                                               END_IF;
                                           END_FOR;
                                           //Beschränkung mögliche Nummer in dem Viereck 5
                                           #initial := 30;
                                           #länge := 32;
                                           FOR #m := 0 TO 2 BY 1 DO
                                               FOR #i := #initial TO #länge BY 1 DO
                                                   IF #gitter[#k].nummer > 0 THEN
                                                       #gitter[#i].potenz_nummer[#gitter[#k].nummer - 1] := FALSE;
                                                   END_IF;
                                               END_FOR;
                                               IF #m < 2 THEN
                                                   #initial := #initial + 9;
                                                   #länge := #länge + 9;
                                               END_IF;
                                           END_FOR;
                                       END_REGION
                                       //Feldchen 41
                                   40:
                                       REGION Feldchen 41
                                           //Beschränkung mögliche Nummer in der Zeile 5
                                           FOR #i := 36 TO 44 BY 1 DO
                                               IF #gitter[#k].nummer > 0 THEN
                                                   #gitter[#i].potenz_nummer[#gitter[#k].nummer - 1] := FALSE;
                                               END_IF;
                                           END_FOR;
                                           //Beschränkung mögliche Nummer in der Säule 5
                                           FOR #i := 4 TO 80 BY 9 DO
                                               IF #gitter[#k].nummer > 0 THEN
                                                   #gitter[#i].potenz_nummer[#gitter[#k].nummer - 1] := FALSE;
                                               END_IF;
                                           END_FOR;
                                           //Beschränkung mögliche Nummer in dem Viereck 5
                                           #initial := 30;
                                           #länge := 32;
                                           FOR #m := 0 TO 2 BY 1 DO
                                               FOR #i := #initial TO #länge BY 1 DO
                                                   IF #gitter[#k].nummer > 0 THEN
                                                       #gitter[#i].potenz_nummer[#gitter[#k].nummer - 1] := FALSE;
                                                   END_IF;
                                               END_FOR;
                                               IF #m < 2 THEN
                                                   #initial := #initial + 9;
                                                   #länge := #länge + 9;
                                               END_IF;
                                           END_FOR;
                                       END_REGION
                                       //Feldchen 42
                                   41:
                                       REGION Feldchen 42
                                           //Beschränkung mögliche Nummer in der Zeile 5
                                           FOR #i := 36 TO 44 BY 1 DO
                                               IF #gitter[#k].nummer > 0 THEN
                                                   #gitter[#i].potenz_nummer[#gitter[#k].nummer - 1] := FALSE;
                                               END_IF;
                                           END_FOR;
                                           //Beschränkung mögliche Nummer in der Säule 6
                                           FOR #i := 5 TO 80 BY 9 DO
                                               IF #gitter[#k].nummer > 0 THEN
                                                   #gitter[#i].potenz_nummer[#gitter[#k].nummer - 1] := FALSE;
                                               END_IF;
                                           END_FOR;
                                           //Beschränkung mögliche Nummer in dem Viereck 5
                                           #initial := 30;
                                           #länge := 32;
                                           FOR #m := 0 TO 2 BY 1 DO
                                               FOR #i := #initial TO #länge BY 1 DO
                                                   IF #gitter[#k].nummer > 0 THEN
                                                       #gitter[#i].potenz_nummer[#gitter[#k].nummer - 1] := FALSE;
                                                   END_IF;
                                               END_FOR;
                                               IF #m < 2 THEN
                                                   #initial := #initial + 9;
                                                   #länge := #länge + 9;
                                               END_IF;
                                           END_FOR;
                                       END_REGION
                                       //Feldchen 43
                                   42:
                                       REGION Feldchen 43
                                           //Beschränkung mögliche Nummer in der Zeile 5
                                           FOR #i := 36 TO 44 BY 1 DO
                                               IF #gitter[#k].nummer > 0 THEN
                                                   #gitter[#i].potenz_nummer[#gitter[#k].nummer - 1] := FALSE;
                                               END_IF;
                                           END_FOR;
                                           //Beschränkung mögliche Nummer in der Säule 7
                                           FOR #i := 6 TO 80 BY 9 DO
                                               IF #gitter[#k].nummer > 0 THEN
                                                   #gitter[#i].potenz_nummer[#gitter[#k].nummer - 1] := FALSE;
                                               END_IF;
                                           END_FOR;
                                           //Beschränkung mögliche Nummer in dem Viereck 6
                                           #initial := 33;
                                           #länge := 35;
                                           FOR #m := 0 TO 2 BY 1 DO
                                               FOR #i := #initial TO #länge BY 1 DO
                                                   IF #gitter[#k].nummer > 0 THEN
                                                       #gitter[#i].potenz_nummer[#gitter[#k].nummer - 1] := FALSE;
                                                   END_IF;
                                               END_FOR;
                                               IF #m < 2 THEN
                                                   #initial := #initial + 9;
                                                   #länge := #länge + 9;
                                               END_IF;
                                           END_FOR;
                                       END_REGION
                                       //Feldchen 44
                                   43:
                                       REGION Feldchen 44
                                           //Beschränkung mögliche Nummer in der Zeile 5
                                           FOR #i := 36 TO 44 BY 1 DO
                                               IF #gitter[#k].nummer > 0 THEN
                                                   #gitter[#i].potenz_nummer[#gitter[#k].nummer - 1] := FALSE;
                                               END_IF;
                                           END_FOR;
                                           //Beschränkung mögliche Nummer in der Säule 8
                                           FOR #i := 7 TO 80 BY 9 DO
                                               IF #gitter[#k].nummer > 0 THEN
                                                   #gitter[#i].potenz_nummer[#gitter[#k].nummer - 1] := FALSE;
                                               END_IF;
                                           END_FOR;
                                           //Beschränkung mögliche Nummer in dem Viereck 6
                                           #initial := 33;
                                           #länge := 35;
                                           FOR #m := 0 TO 2 BY 1 DO
                                               FOR #i := #initial TO #länge BY 1 DO
                                                   IF #gitter[#k].nummer > 0 THEN
                                                       #gitter[#i].potenz_nummer[#gitter[#k].nummer - 1] := FALSE;
                                                   END_IF;
                                               END_FOR;
                                               IF #m < 2 THEN
                                                   #initial := #initial + 9;
                                                   #länge := #länge + 9;
                                               END_IF;
                                           END_FOR;
                                       END_REGION
                                       //Feldchen 45
                                   44:
                                       REGION Feldchen 45
                                           //Beschränkung mögliche Nummer in der Zeile 5
                                           FOR #i := 36 TO 44 BY 1 DO
                                               IF #gitter[#k].nummer > 0 THEN
                                                   #gitter[#i].potenz_nummer[#gitter[#k].nummer - 1] := FALSE;
                                               END_IF;
                                           END_FOR;
                                           //Beschränkung mögliche Nummer in der Säule 9
                                           FOR #i := 8 TO 80 BY 9 DO
                                               IF #gitter[#k].nummer > 0 THEN
                                                   #gitter[#i].potenz_nummer[#gitter[#k].nummer - 1] := FALSE;
                                               END_IF;
                                           END_FOR;
                                           //Beschränkung mögliche Nummer in dem Viereck 6
                                           #initial := 33;
                                           #länge := 35;
                                           FOR #m := 0 TO 2 BY 1 DO
                                               FOR #i := #initial TO #länge BY 1 DO
                                                   IF #gitter[#k].nummer > 0 THEN
                                                       #gitter[#i].potenz_nummer[#gitter[#k].nummer - 1] := FALSE;
                                                   END_IF;
                                               END_FOR;
                                               IF #m < 2 THEN
                                                   #initial := #initial + 9;
                                                   #länge := #länge + 9;
                                               END_IF;
                                           END_FOR;
                                       END_REGION
                                       //Feldchen 46
                                   45:
                                       REGION Feldchen 46
                                           //Beschränkung mögliche Nummer in der Zeile 6
                                           FOR #i := 45 TO 53 BY 1 DO
                                               IF #gitter[#k].nummer > 0 THEN
                                                   #gitter[#i].potenz_nummer[#gitter[#k].nummer - 1] := FALSE;
                                               END_IF;
                                           END_FOR;
                                           //Beschränkung mögliche Nummer in der Säule 1
                                           FOR #i := 0 TO 80 BY 9 DO
                                               IF #gitter[#k].nummer > 0 THEN
                                                   #gitter[#i].potenz_nummer[#gitter[#k].nummer - 1] := FALSE;
                                               END_IF;
                                           END_FOR;
                                           //Beschränkung mögliche Nummer in dem Viereck 4
                                           #initial := 27;
                                           #länge := 29;
                                           FOR #m := 0 TO 2 BY 1 DO
                                               FOR #i := #initial TO #länge BY 1 DO
                                                   IF #gitter[#k].nummer > 0 THEN
                                                       #gitter[#i].potenz_nummer[#gitter[#k].nummer - 1] := FALSE;
                                                   END_IF;
                                               END_FOR;
                                               IF #m < 2 THEN
                                                   #initial := #initial + 9;
                                                   #länge := #länge + 9;
                                               END_IF;
                                           END_FOR;
                                       END_REGION
                                       //Feldchen 47
                                   46:
                                       REGION Feldchen 47
                                           //Beschränkung mögliche Nummer in der Zeile 6
                                           FOR #i := 45 TO 53 BY 1 DO
                                               IF #gitter[#k].nummer > 0 THEN
                                                   #gitter[#i].potenz_nummer[#gitter[#k].nummer - 1] := FALSE;
                                               END_IF;
                                           END_FOR;
                                           //Beschränkung mögliche Nummer in der Säule 2
                                           FOR #i := 1 TO 80 BY 9 DO
                                               IF #gitter[#k].nummer > 0 THEN
                                                   #gitter[#i].potenz_nummer[#gitter[#k].nummer - 1] := FALSE;
                                               END_IF;
                                           END_FOR;
                                           //Beschränkung mögliche Nummer in dem Viereck 4
                                           #initial := 27;
                                           #länge := 29;
                                           FOR #m := 0 TO 2 BY 1 DO
                                               FOR #i := #initial TO #länge BY 1 DO
                                                   IF #gitter[#k].nummer > 0 THEN
                                                       #gitter[#i].potenz_nummer[#gitter[#k].nummer - 1] := FALSE;
                                                   END_IF;
                                               END_FOR;
                                               IF #m < 2 THEN
                                                   #initial := #initial + 9;
                                                   #länge := #länge + 9;
                                               END_IF;
                                           END_FOR;
                                       END_REGION
                                       //Feldchen 48
                                   47:
                                       REGION Feldchen 48
                                           //Beschränkung mögliche Nummer in der Zeile 6
                                           FOR #i := 45 TO 53 BY 1 DO
                                               IF #gitter[#k].nummer > 0 THEN
                                                   #gitter[#i].potenz_nummer[#gitter[#k].nummer - 1] := FALSE;
                                               END_IF;
                                           END_FOR;
                                           //Beschränkung mögliche Nummer in der Säule 3
                                           FOR #i := 2 TO 80 BY 9 DO
                                               IF #gitter[#k].nummer > 0 THEN
                                                   #gitter[#i].potenz_nummer[#gitter[#k].nummer - 1] := FALSE;
                                               END_IF;
                                           END_FOR;
                                           //Beschränkung mögliche Nummer in dem Viereck 4
                                           #initial := 27;
                                           #länge := 29;
                                           FOR #m := 0 TO 2 BY 1 DO
                                               FOR #i := #initial TO #länge BY 1 DO
                                                   IF #gitter[#k].nummer > 0 THEN
                                                       #gitter[#i].potenz_nummer[#gitter[#k].nummer - 1] := FALSE;
                                                   END_IF;
                                               END_FOR;
                                               IF #m < 2 THEN
                                                   #initial := #initial + 9;
                                                   #länge := #länge + 9;
                                               END_IF;
                                           END_FOR;
                                       END_REGION
                                       //Feldchen 49
                                   48:
                                       REGION Feldchen 49
                                           //Beschränkung mögliche Nummer in der Zeile 6
                                           FOR #i := 45 TO 53 BY 1 DO
                                               IF #gitter[#k].nummer > 0 THEN
                                                   #gitter[#i].potenz_nummer[#gitter[#k].nummer - 1] := FALSE;
                                               END_IF;
                                           END_FOR;
                                           //Beschränkung mögliche Nummer in der Säule 4
                                           FOR #i := 3 TO 80 BY 9 DO
                                               IF #gitter[#k].nummer > 0 THEN
                                                   #gitter[#i].potenz_nummer[#gitter[#k].nummer - 1] := FALSE;
                                               END_IF;
                                           END_FOR;
                                           //Beschränkung mögliche Nummer in dem Viereck 5
                                           #initial := 30;
                                           #länge := 32;
                                           FOR #m := 0 TO 2 BY 1 DO
                                               FOR #i := #initial TO #länge BY 1 DO
                                                   IF #gitter[#k].nummer > 0 THEN
                                                       #gitter[#i].potenz_nummer[#gitter[#k].nummer - 1] := FALSE;
                                                   END_IF;
                                               END_FOR;
                                               IF #m < 2 THEN
                                                   #initial := #initial + 9;
                                                   #länge := #länge + 9;
                                               END_IF;
                                           END_FOR;
                                       END_REGION
                                       //Feldchen 50
                                   49:
                                       REGION Feldchen 50
                                           //Beschränkung mögliche Nummer in der Zeile 6
                                           FOR #i := 45 TO 53 BY 1 DO
                                               IF #gitter[#k].nummer > 0 THEN
                                                   #gitter[#i].potenz_nummer[#gitter[#k].nummer - 1] := FALSE;
                                               END_IF;
                                           END_FOR;
                                           //Beschränkung mögliche Nummer in der Säule 5
                                           FOR #i := 4 TO 80 BY 9 DO
                                               IF #gitter[#k].nummer > 0 THEN
                                                   #gitter[#i].potenz_nummer[#gitter[#k].nummer - 1] := FALSE;
                                               END_IF;
                                           END_FOR;
                                           //Beschränkung mögliche Nummer in dem Viereck 5
                                           #initial := 30;
                                           #länge := 32;
                                           FOR #m := 0 TO 2 BY 1 DO
                                               FOR #i := #initial TO #länge BY 1 DO
                                                   IF #gitter[#k].nummer > 0 THEN
                                                       #gitter[#i].potenz_nummer[#gitter[#k].nummer - 1] := FALSE;
                                                   END_IF;
                                               END_FOR;
                                               IF #m < 2 THEN
                                                   #initial := #initial + 9;
                                                   #länge := #länge + 9;
                                               END_IF;
                                           END_FOR;
                                       END_REGION
                                       //Feldchen 51
                                   50:
                                       REGION Feldchen 51
                                           //Beschränkung mögliche Nummer in der Zeile 6
                                           FOR #i := 45 TO 53 BY 1 DO
                                               IF #gitter[#k].nummer > 0 THEN
                                                   #gitter[#i].potenz_nummer[#gitter[#k].nummer - 1] := FALSE;
                                               END_IF;
                                           END_FOR;
                                           //Beschränkung mögliche Nummer in der Säule 6
                                           FOR #i := 5 TO 80 BY 9 DO
                                               IF #gitter[#k].nummer > 0 THEN
                                                   #gitter[#i].potenz_nummer[#gitter[#k].nummer - 1] := FALSE;
                                               END_IF;
                                           END_FOR;
                                           //Beschränkung mögliche Nummer in dem Viereck 5
                                           #initial := 30;
                                           #länge := 32;
                                           FOR #m := 0 TO 2 BY 1 DO
                                               FOR #i := #initial TO #länge BY 1 DO
                                                   IF #gitter[#k].nummer > 0 THEN
                                                       #gitter[#i].potenz_nummer[#gitter[#k].nummer - 1] := FALSE;
                                                   END_IF;
                                               END_FOR;
                                               IF #m < 2 THEN
                                                   #initial := #initial + 9;
                                                   #länge := #länge + 9;
                                               END_IF;
                                           END_FOR;
                                       END_REGION
                                       //Feldchen 52
                                   51:
                                       REGION Feldchen 52
                                           //Beschränkung mögliche Nummer in der Zeile 6
                                           FOR #i := 45 TO 53 BY 1 DO
                                               IF #gitter[#k].nummer > 0 THEN
                                                   #gitter[#i].potenz_nummer[#gitter[#k].nummer - 1] := FALSE;
                                               END_IF;
                                           END_FOR;
                                           //Beschränkung mögliche Nummer in der Säule 7
                                           FOR #i := 6 TO 80 BY 9 DO
                                               IF #gitter[#k].nummer > 0 THEN
                                                   #gitter[#i].potenz_nummer[#gitter[#k].nummer - 1] := FALSE;
                                               END_IF;
                                           END_FOR;
                                           //Beschränkung mögliche Nummer in dem Viereck 6
                                           #initial := 33;
                                           #länge := 35;
                                           FOR #m := 0 TO 2 BY 1 DO
                                               FOR #i := #initial TO #länge BY 1 DO
                                                   IF #gitter[#k].nummer > 0 THEN
                                                       #gitter[#i].potenz_nummer[#gitter[#k].nummer - 1] := FALSE;
                                                   END_IF;
                                               END_FOR;
                                               IF #m < 2 THEN
                                                   #initial := #initial + 9;
                                                   #länge := #länge + 9;
                                               END_IF;
                                           END_FOR;
                                       END_REGION
                                       //Feldchen 53
                                   52:
                                       REGION Feldchen 53
                                           //Beschränkung mögliche Nummer in der Zeile 6
                                           FOR #i := 45 TO 53 BY 1 DO
                                               IF #gitter[#k].nummer > 0 THEN
                                                   #gitter[#i].potenz_nummer[#gitter[#k].nummer - 1] := FALSE;
                                               END_IF;
                                           END_FOR;
                                           //Beschränkung mögliche Nummer in der Säule 8
                                           FOR #i := 7 TO 80 BY 9 DO
                                               IF #gitter[#k].nummer > 0 THEN
                                                   #gitter[#i].potenz_nummer[#gitter[#k].nummer - 1] := FALSE;
                                               END_IF;
                                           END_FOR;
                                           //Beschränkung mögliche Nummer in dem Viereck 6
                                           #initial := 33;
                                           #länge := 35;
                                           FOR #m := 0 TO 2 BY 1 DO
                                               FOR #i := #initial TO #länge BY 1 DO
                                                   IF #gitter[#k].nummer > 0 THEN
                                                       #gitter[#i].potenz_nummer[#gitter[#k].nummer - 1] := FALSE;
                                                   END_IF;
                                               END_FOR;
                                               IF #m < 2 THEN
                                                   #initial := #initial + 9;
                                                   #länge := #länge + 9;
                                               END_IF;
                                           END_FOR;
                                       END_REGION
                                       //Feldchen 54
                                   53:
                                       REGION Feldchen 54
                                           //Beschränkung mögliche Nummer in der Zeile 6
                                           FOR #i := 45 TO 53 BY 1 DO
                                               IF #gitter[#k].nummer > 0 THEN
                                                   #gitter[#i].potenz_nummer[#gitter[#k].nummer - 1] := FALSE;
                                               END_IF;
                                           END_FOR;
                                           //Beschränkung mögliche Nummer in der Säule 9
                                           FOR #i := 8 TO 80 BY 9 DO
                                               IF #gitter[#k].nummer > 0 THEN
                                                   #gitter[#i].potenz_nummer[#gitter[#k].nummer - 1] := FALSE;
                                               END_IF;
                                           END_FOR;
                                           //Beschränkung mögliche Nummer in dem Viereck 6
                                           #initial := 33;
                                           #länge := 35;
                                           FOR #m := 0 TO 2 BY 1 DO
                                               FOR #i := #initial TO #länge BY 1 DO
                                                   IF #gitter[#k].nummer > 0 THEN
                                                       #gitter[#i].potenz_nummer[#gitter[#k].nummer - 1] := FALSE;
                                                   END_IF;
                                               END_FOR;
                                               IF #m < 2 THEN
                                                   #initial := #initial + 9;
                                                   #länge := #länge + 9;
                                               END_IF;
                                           END_FOR;
                                       END_REGION
                                       //Feldchen 55
                                   54:
                                       REGION Feldchen 55
                                           //Beschränkung mögliche Nummer in der Zeile 7
                                           FOR #i := 54 TO 62 BY 1 DO
                                               IF #gitter[#k].nummer > 0 THEN
                                                   #gitter[#i].potenz_nummer[#gitter[#k].nummer - 1] := FALSE;
                                               END_IF;
                                           END_FOR;
                                           //Beschränkung mögliche Nummer in der Säule 1
                                           FOR #i := 0 TO 80 BY 9 DO
                                               IF #gitter[#k].nummer > 0 THEN
                                                   #gitter[#i].potenz_nummer[#gitter[#k].nummer - 1] := FALSE;
                                               END_IF;
                                           END_FOR;
                                           //Beschränkung mögliche Nummer in dem Viereck 7
                                           #initial := 54;
                                           #länge := 56;
                                           FOR #m := 0 TO 2 BY 1 DO
                                               FOR #i := #initial TO #länge BY 1 DO
                                                   IF #gitter[#k].nummer > 0 THEN
                                                       #gitter[#i].potenz_nummer[#gitter[#k].nummer - 1] := FALSE;
                                                   END_IF;
                                               END_FOR;
                                               IF #m < 2 THEN
                                                   #initial := #initial + 9;
                                                   #länge := #länge + 9;
                                               END_IF;
                                           END_FOR;
                                       END_REGION
                                       //Feldchen 56
                                   55:
                                       REGION Feldchen 56
                                           //Beschränkung mögliche Nummer in der Zeile 7
                                           FOR #i := 54 TO 62 BY 1 DO
                                               IF #gitter[#k].nummer > 0 THEN
                                                   #gitter[#i].potenz_nummer[#gitter[#k].nummer - 1] := FALSE;
                                               END_IF;
                                           END_FOR;
                                           //Beschränkung mögliche Nummer in der Säule 2
                                           FOR #i := 1 TO 80 BY 9 DO
                                               IF #gitter[#k].nummer > 0 THEN
                                                   #gitter[#i].potenz_nummer[#gitter[#k].nummer - 1] := FALSE;
                                               END_IF;
                                           END_FOR;
                                           //Beschränkung mögliche Nummer in dem Viereck 7
                                           #initial := 54;
                                           #länge := 56;
                                           FOR #m := 0 TO 2 BY 1 DO
                                               FOR #i := #initial TO #länge BY 1 DO
                                                   IF #gitter[#k].nummer > 0 THEN
                                                       #gitter[#i].potenz_nummer[#gitter[#k].nummer - 1] := FALSE;
                                                   END_IF;
                                               END_FOR;
                                               IF #m < 2 THEN
                                                   #initial := #initial + 9;
                                                   #länge := #länge + 9;
                                               END_IF;
                                           END_FOR;
                                       END_REGION
                                       //Feldchen 57
                                   56:
                                       REGION Feldchen 57
                                           //Beschränkung mögliche Nummer in der Zeile 7
                                           FOR #i := 54 TO 62 BY 1 DO
                                               IF #gitter[#k].nummer > 0 THEN
                                                   #gitter[#i].potenz_nummer[#gitter[#k].nummer - 1] := FALSE;
                                               END_IF;
                                           END_FOR;
                                           //Beschränkung mögliche Nummer in der Säule 3
                                           FOR #i := 2 TO 80 BY 9 DO
                                               IF #gitter[#k].nummer > 0 THEN
                                                   #gitter[#i].potenz_nummer[#gitter[#k].nummer - 1] := FALSE;
                                               END_IF;
                                           END_FOR;
                                           //Beschränkung mögliche Nummer in dem Viereck 7
                                           #initial := 54;
                                           #länge := 56;
                                           FOR #m := 0 TO 2 BY 1 DO
                                               FOR #i := #initial TO #länge BY 1 DO
                                                   IF #gitter[#k].nummer > 0 THEN
                                                       #gitter[#i].potenz_nummer[#gitter[#k].nummer - 1] := FALSE;
                                                   END_IF;
                                               END_FOR;
                                               IF #m < 2 THEN
                                                   #initial := #initial + 9;
                                                   #länge := #länge + 9;
                                               END_IF;
                                           END_FOR;
                                       END_REGION //Feldchen 57
                                       //Feldchen 58
                                   57:
                                       REGION Feldchen 58
                                           //Beschränkung mögliche Nummer in der Zeile 7
                                           FOR #i := 54 TO 62 BY 1 DO
                                               IF #gitter[#k].nummer > 0 THEN
                                                   #gitter[#i].potenz_nummer[#gitter[#k].nummer - 1] := FALSE;
                                               END_IF;
                                           END_FOR;
                                           //Beschränkung mögliche Nummer in der Säule 4
                                           FOR #i := 3 TO 80 BY 9 DO
                                               IF #gitter[#k].nummer > 0 THEN
                                                   #gitter[#i].potenz_nummer[#gitter[#k].nummer - 1] := FALSE;
                                               END_IF;
                                           END_FOR;
                                           //Beschränkung mögliche Nummer in dem Viereck 8
                                           #initial := 57;
                                           #länge := 59;
                                           FOR #m := 0 TO 2 BY 1 DO
                                               FOR #i := #initial TO #länge BY 1 DO
                                                   IF #gitter[#k].nummer > 0 THEN
                                                       #gitter[#i].potenz_nummer[#gitter[#k].nummer - 1] := FALSE;
                                                   END_IF;
                                               END_FOR;
                                               IF #m < 2 THEN
                                                   #initial := #initial + 9;
                                                   #länge := #länge + 9;
                                               END_IF;
                                           END_FOR;
                                       END_REGION
                                       //Feldchen 59
                                   58:
                                       REGION Feldchen 59
                                           //Beschränkung mögliche Nummer in der Zeile 7
                                           FOR #i := 54 TO 62 BY 1 DO
                                               IF #gitter[#k].nummer > 0 THEN
                                                   #gitter[#i].potenz_nummer[#gitter[#k].nummer - 1] := FALSE;
                                               END_IF;
                                           END_FOR;
                                           //Beschränkung mögliche Nummer in der Säule 5
                                           FOR #i := 4 TO 80 BY 9 DO
                                               IF #gitter[#k].nummer > 0 THEN
                                                   #gitter[#i].potenz_nummer[#gitter[#k].nummer - 1] := FALSE;
                                               END_IF;
                                           END_FOR;
                                           //Beschränkung mögliche Nummer in dem Viereck 8
                                           #initial := 57;
                                           #länge := 59;
                                           FOR #m := 0 TO 2 BY 1 DO
                                               FOR #i := #initial TO #länge BY 1 DO
                                                   IF #gitter[#k].nummer > 0 THEN
                                                       #gitter[#i].potenz_nummer[#gitter[#k].nummer - 1] := FALSE;
                                                   END_IF;
                                               END_FOR;
                                               IF #m < 2 THEN
                                                   #initial := #initial + 9;
                                                   #länge := #länge + 9;
                                               END_IF;
                                           END_FOR;
                                       END_REGION
                                       //Feldchen 60
                                   59:
                                       REGION Feldchen 60
                                           //Beschränkung mögliche Nummer in der Zeile 7
                                           FOR #i := 54 TO 62 BY 1 DO
                                               IF #gitter[#k].nummer > 0 THEN
                                                   #gitter[#i].potenz_nummer[#gitter[#k].nummer - 1] := FALSE;
                                               END_IF;
                                           END_FOR;
                                           //Beschränkung mögliche Nummer in der Säule 6
                                           FOR #i := 5 TO 80 BY 9 DO
                                               IF #gitter[#k].nummer > 0 THEN
                                                   #gitter[#i].potenz_nummer[#gitter[#k].nummer - 1] := FALSE;
                                               END_IF;
                                           END_FOR;
                                           //Beschränkung mögliche Nummer in dem Viereck 8
                                           #initial := 57;
                                           #länge := 59;
                                           FOR #m := 0 TO 2 BY 1 DO
                                               FOR #i := #initial TO #länge BY 1 DO
                                                   IF #gitter[#k].nummer > 0 THEN
                                                       #gitter[#i].potenz_nummer[#gitter[#k].nummer - 1] := FALSE;
                                                   END_IF;
                                               END_FOR;
                                               IF #m < 2 THEN
                                                   #initial := #initial + 9;
                                                   #länge := #länge + 9;
                                               END_IF;
                                           END_FOR;
                                       END_REGION
                                       //Feldchen 61
                                   60:
                                       REGION Feldchen 61
                                           //Beschränkung mögliche Nummer in der Zeile 7
                                           FOR #i := 54 TO 62 BY 1 DO
                                               IF #gitter[#k].nummer > 0 THEN
                                                   #gitter[#i].potenz_nummer[#gitter[#k].nummer - 1] := FALSE;
                                               END_IF;
                                           END_FOR;
                                           //Beschränkung mögliche Nummer in der Säule 7
                                           FOR #i := 6 TO 80 BY 9 DO
                                               IF #gitter[#k].nummer > 0 THEN
                                                   #gitter[#i].potenz_nummer[#gitter[#k].nummer - 1] := FALSE;
                                               END_IF;
                                           END_FOR;
                                           //Beschränkung mögliche Nummer in dem Viereck 9
                                           #initial := 60;
                                           #länge := 62;
                                           FOR #m := 0 TO 2 BY 1 DO
                                               FOR #i := #initial TO #länge BY 1 DO
                                                   IF #gitter[#k].nummer > 0 THEN
                                                       #gitter[#i].potenz_nummer[#gitter[#k].nummer - 1] := FALSE;
                                                   END_IF;
                                               END_FOR;
                                               IF #m < 2 THEN
                                                   #initial := #initial + 9;
                                                   #länge := #länge + 9;
                                               END_IF;
                                           END_FOR;
                                       END_REGION
                                       //Feldchen 62
                                   61:
                                       REGION Feldchen 62
                                           //Beschränkung mögliche Nummer in der Zeile 7
                                           FOR #i := 54 TO 62 BY 1 DO
                                               IF #gitter[#k].nummer > 0 THEN
                                                   #gitter[#i].potenz_nummer[#gitter[#k].nummer - 1] := FALSE;
                                               END_IF;
                                           END_FOR;
                                           //Beschränkung mögliche Nummer in der Säule 8
                                           FOR #i := 7 TO 80 BY 9 DO
                                               IF #gitter[#k].nummer > 0 THEN
                                                   #gitter[#i].potenz_nummer[#gitter[#k].nummer - 1] := FALSE;
                                               END_IF;
                                           END_FOR;
                                           //Beschränkung mögliche Nummer in dem Viereck 9
                                           #initial := 60;
                                           #länge := 62;
                                           FOR #m := 0 TO 2 BY 1 DO
                                               FOR #i := #initial TO #länge BY 1 DO
                                                   IF #gitter[#k].nummer > 0 THEN
                                                       #gitter[#i].potenz_nummer[#gitter[#k].nummer - 1] := FALSE;
                                                   END_IF;
                                               END_FOR;
                                               IF #m < 2 THEN
                                                   #initial := #initial + 9;
                                                   #länge := #länge + 9;
                                               END_IF;
                                           END_FOR;
                                       END_REGION
                                       //Feldchen 63
                                   62:
                                       REGION Feldchen 63
                                           //Beschränkung mögliche Nummer in der Zeile 7
                                           FOR #i := 54 TO 62 BY 1 DO
                                               IF #gitter[#k].nummer > 0 THEN
                                                   #gitter[#i].potenz_nummer[#gitter[#k].nummer - 1] := FALSE;
                                               END_IF;
                                           END_FOR;
                                           //Beschränkung mögliche Nummer in der Säule 9
                                           FOR #i := 8 TO 80 BY 9 DO
                                               IF #gitter[#k].nummer > 0 THEN
                                                   #gitter[#i].potenz_nummer[#gitter[#k].nummer - 1] := FALSE;
                                               END_IF;
                                           END_FOR;
                                           //Beschränkung mögliche Nummer in dem Viereck 9
                                           #initial := 60;
                                           #länge := 62;
                                           FOR #m := 0 TO 2 BY 1 DO
                                               FOR #i := #initial TO #länge BY 1 DO
                                                   IF #gitter[#k].nummer > 0 THEN
                                                       #gitter[#i].potenz_nummer[#gitter[#k].nummer - 1] := FALSE;
                                                   END_IF;
                                               END_FOR;
                                               IF #m < 2 THEN
                                                   #initial := #initial + 9;
                                                   #länge := #länge + 9;
                                               END_IF;
                                           END_FOR;
                                       END_REGION
                                       //Feldchen 64
                                   63:
                                       REGION Feldchen 64
                                           //Beschränkung mögliche Nummer in der Zeile 8
                                           FOR #i := 63 TO 71 BY 1 DO
                                               IF #gitter[#k].nummer > 0 THEN
                                                   #gitter[#i].potenz_nummer[#gitter[#k].nummer - 1] := FALSE;
                                               END_IF;
                                           END_FOR;
                                           //Beschränkung mögliche Nummer in der Säule 1
                                           FOR #i := 0 TO 80 BY 9 DO
                                               IF #gitter[#k].nummer > 0 THEN
                                                   #gitter[#i].potenz_nummer[#gitter[#k].nummer - 1] := FALSE;
                                               END_IF;
                                           END_FOR;
                                           //Beschränkung mögliche Nummer in dem Viereck 7
                                           #initial := 54;
                                           #länge := 56;
                                           FOR #m := 0 TO 2 BY 1 DO
                                               FOR #i := #initial TO #länge BY 1 DO
                                                   IF #gitter[#k].nummer > 0 THEN
                                                       #gitter[#i].potenz_nummer[#gitter[#k].nummer - 1] := FALSE;
                                                   END_IF;
                                               END_FOR;
                                               IF #m < 2 THEN
                                                   #initial := #initial + 9;
                                                   #länge := #länge + 9;
                                               END_IF;
                                           END_FOR;
                                       END_REGION
                                       //Feldchen 65
                                   64:
                                       REGION Feldchen 65
                                           //Beschränkung mögliche Nummer in der Zeile 8
                                           FOR #i := 63 TO 71 BY 1 DO
                                               IF #gitter[#k].nummer > 0 THEN
                                                   #gitter[#i].potenz_nummer[#gitter[#k].nummer - 1] := FALSE;
                                               END_IF;
                                           END_FOR;
                                           //Beschränkung mögliche Nummer in der Säule 2
                                           FOR #i := 1 TO 80 BY 9 DO
                                               IF #gitter[#k].nummer > 0 THEN
                                                   #gitter[#i].potenz_nummer[#gitter[#k].nummer - 1] := FALSE;
                                               END_IF;
                                           END_FOR;
                                           //Beschränkung mögliche Nummer in dem Viereck 7
                                           #initial := 54;
                                           #länge := 56;
                                           FOR #m := 0 TO 2 BY 1 DO
                                               FOR #i := #initial TO #länge BY 1 DO
                                                   IF #gitter[#k].nummer > 0 THEN
                                                       #gitter[#i].potenz_nummer[#gitter[#k].nummer - 1] := FALSE;
                                                   END_IF;
                                               END_FOR;
                                               IF #m < 2 THEN
                                                   #initial := #initial + 9;
                                                   #länge := #länge + 9;
                                               END_IF;
                                           END_FOR;
                                       END_REGION
                                       //Feldchen 66
                                   65:
                                       REGION Feldchen 66
                                           //Beschränkung mögliche Nummer in der Zeile 8
                                           FOR #i := 63 TO 71 BY 1 DO
                                               IF #gitter[#k].nummer > 0 THEN
                                                   #gitter[#i].potenz_nummer[#gitter[#k].nummer - 1] := FALSE;
                                               END_IF;
                                           END_FOR;
                                           //Beschränkung mögliche Nummer in der Säule 3
                                           FOR #i := 2 TO 80 BY 9 DO
                                               IF #gitter[#k].nummer > 0 THEN
                                                   #gitter[#i].potenz_nummer[#gitter[#k].nummer - 1] := FALSE;
                                               END_IF;
                                           END_FOR;
                                           //Beschränkung mögliche Nummer in dem Viereck 7
                                           #initial := 54;
                                           #länge := 56;
                                           FOR #m := 0 TO 2 BY 1 DO
                                               FOR #i := #initial TO #länge BY 1 DO
                                                   IF #gitter[#k].nummer > 0 THEN
                                                       #gitter[#i].potenz_nummer[#gitter[#k].nummer - 1] := FALSE;
                                                   END_IF;
                                               END_FOR;
                                               IF #m < 2 THEN
                                                   #initial := #initial + 9;
                                                   #länge := #länge + 9;
                                               END_IF;
                                           END_FOR;
                                       END_REGION
                                       //Feldchen 67
                                   66:
                                       REGION Feldchen 67
                                           //Beschränkung mögliche Nummer in der Zeile 8
                                           FOR #i := 63 TO 71 BY 1 DO
                                               IF #gitter[#k].nummer > 0 THEN
                                                   #gitter[#i].potenz_nummer[#gitter[#k].nummer - 1] := FALSE;
                                               END_IF;
                                           END_FOR;
                                           //Beschränkung mögliche Nummer in der Säule 4
                                           FOR #i := 3 TO 80 BY 9 DO
                                               IF #gitter[#k].nummer > 0 THEN
                                                   #gitter[#i].potenz_nummer[#gitter[#k].nummer - 1] := FALSE;
                                               END_IF;
                                           END_FOR;
                                           //Beschränkung mögliche Nummer in dem Viereck 8
                                           #initial := 57;
                                           #länge := 59;
                                           FOR #m := 0 TO 2 BY 1 DO
                                               FOR #i := #initial TO #länge BY 1 DO
                                                   IF #gitter[#k].nummer > 0 THEN
                                                       #gitter[#i].potenz_nummer[#gitter[#k].nummer - 1] := FALSE;
                                                   END_IF;
                                               END_FOR;
                                               IF #m < 2 THEN
                                                   #initial := #initial + 9;
                                                   #länge := #länge + 9;
                                               END_IF;
                                           END_FOR;
                                       END_REGION
                                       //Feldchen 68
                                   67:
                                       REGION Feldchen 68
                                           //Beschränkung mögliche Nummer in der Zeile 8
                                           FOR #i := 63 TO 71 BY 1 DO
                                               IF #gitter[#k].nummer > 0 THEN
                                                   #gitter[#i].potenz_nummer[#gitter[#k].nummer - 1] := FALSE;
                                               END_IF;
                                           END_FOR;
                                           //Beschränkung mögliche Nummer in der Säule 5
                                           FOR #i := 4 TO 80 BY 9 DO
                                               IF #gitter[#k].nummer > 0 THEN
                                                   #gitter[#i].potenz_nummer[#gitter[#k].nummer - 1] := FALSE;
                                               END_IF;
                                           END_FOR;
                                           //Beschränkung mögliche Nummer in dem Viereck 8
                                           #initial := 57;
                                           #länge := 59;
                                           FOR #m := 0 TO 2 BY 1 DO
                                               FOR #i := #initial TO #länge BY 1 DO
                                                   IF #gitter[#k].nummer > 0 THEN
                                                       #gitter[#i].potenz_nummer[#gitter[#k].nummer - 1] := FALSE;
                                                   END_IF;
                                               END_FOR;
                                               IF #m < 2 THEN
                                                   #initial := #initial + 9;
                                                   #länge := #länge + 9;
                                               END_IF;
                                           END_FOR;
                                       END_REGION
                                       //Feldchen 69
                                   68:
                                       REGION Feldchen 69
                                           //Beschränkung mögliche Nummer in der Zeile 8
                                           FOR #i := 63 TO 71 BY 1 DO
                                               IF #gitter[#k].nummer > 0 THEN
                                                   #gitter[#i].potenz_nummer[#gitter[#k].nummer - 1] := FALSE;
                                               END_IF;
                                           END_FOR;
                                           //Beschränkung mögliche Nummer in der Säule 6
                                           FOR #i := 5 TO 80 BY 9 DO
                                               IF #gitter[#k].nummer > 0 THEN
                                                   #gitter[#i].potenz_nummer[#gitter[#k].nummer - 1] := FALSE;
                                               END_IF;
                                           END_FOR;
                                           //Beschränkung mögliche Nummer in dem Viereck 8
                                           #initial := 57;
                                           #länge := 59;
                                           FOR #m := 0 TO 2 BY 1 DO
                                               FOR #i := #initial TO #länge BY 1 DO
                                                   IF #gitter[#k].nummer > 0 THEN
                                                       #gitter[#i].potenz_nummer[#gitter[#k].nummer - 1] := FALSE;
                                                   END_IF;
                                               END_FOR;
                                               IF #m < 2 THEN
                                                   #initial := #initial + 9;
                                                   #länge := #länge + 9;
                                               END_IF;
                                           END_FOR;
                                       END_REGION
                                       //Feldchen 70
                                   69:
                                       REGION Feldchen 70
                                           //Beschränkung mögliche Nummer in der Zeile 8
                                           FOR #i := 63 TO 71 BY 1 DO
                                               IF #gitter[#k].nummer > 0 THEN
                                                   #gitter[#i].potenz_nummer[#gitter[#k].nummer - 1] := FALSE;
                                               END_IF;
                                           END_FOR;
                                           //Beschränkung mögliche Nummer in der Säule 7
                                           FOR #i := 6 TO 80 BY 9 DO
                                               IF #gitter[#k].nummer > 0 THEN
                                                   #gitter[#i].potenz_nummer[#gitter[#k].nummer - 1] := FALSE;
                                               END_IF;
                                           END_FOR;
                                           //Beschränkung mögliche Nummer in dem Viereck 9
                                           #initial := 60;
                                           #länge := 62;
                                           FOR #m := 0 TO 2 BY 1 DO
                                               FOR #i := #initial TO #länge BY 1 DO
                                                   IF #gitter[#k].nummer > 0 THEN
                                                       #gitter[#i].potenz_nummer[#gitter[#k].nummer - 1] := FALSE;
                                                   END_IF;
                                               END_FOR;
                                               IF #m < 2 THEN
                                                   #initial := #initial + 9;
                                                   #länge := #länge + 9;
                                               END_IF;
                                           END_FOR;
                                       END_REGION
                                       //Feldchen 71
                                   70:
                                       REGION Feldchen 71
                                           //Beschränkung mögliche Nummer in der Zeile 8
                                           FOR #i := 63 TO 71 BY 1 DO
                                               IF #gitter[#k].nummer > 0 THEN
                                                   #gitter[#i].potenz_nummer[#gitter[#k].nummer - 1] := FALSE;
                                               END_IF;
                                           END_FOR;
                                           //Beschränkung mögliche Nummer in der Säule 8
                                           FOR #i := 7 TO 80 BY 9 DO
                                               IF #gitter[#k].nummer > 0 THEN
                                                   #gitter[#i].potenz_nummer[#gitter[#k].nummer - 1] := FALSE;
                                               END_IF;
                                           END_FOR;
                                           //Beschränkung mögliche Nummer in dem Viereck 9
                                           #initial := 60;
                                           #länge := 62;
                                           FOR #m := 0 TO 2 BY 1 DO
                                               FOR #i := #initial TO #länge BY 1 DO
                                                   IF #gitter[#k].nummer > 0 THEN
                                                       #gitter[#i].potenz_nummer[#gitter[#k].nummer - 1] := FALSE;
                                                   END_IF;
                                               END_FOR;
                                               IF #m < 2 THEN
                                                   #initial := #initial + 9;
                                                   #länge := #länge + 9;
                                               END_IF;
                                           END_FOR;
                                       END_REGION
                                       //Feldchen 72
                                   71:
                                       REGION Feldchen 72
                                           //Beschränkung mögliche Nummer in der Zeile 8
                                           FOR #i := 63 TO 71 BY 1 DO
                                               IF #gitter[#k].nummer > 0 THEN
                                                   #gitter[#i].potenz_nummer[#gitter[#k].nummer - 1] := FALSE;
                                               END_IF;
                                           END_FOR;
                                           //Beschränkung mögliche Nummer in der Säule 9
                                           FOR #i := 8 TO 80 BY 9 DO
                                               IF #gitter[#k].nummer > 0 THEN
                                                   #gitter[#i].potenz_nummer[#gitter[#k].nummer - 1] := FALSE;
                                               END_IF;
                                           END_FOR;
                                           //Beschränkung mögliche Nummer in dem Viereck 9
                                           #initial := 60;
                                           #länge := 62;
                                           FOR #m := 0 TO 2 BY 1 DO
                                               FOR #i := #initial TO #länge BY 1 DO
                                                   IF #gitter[#k].nummer > 0 THEN
                                                       #gitter[#i].potenz_nummer[#gitter[#k].nummer - 1] := FALSE;
                                                   END_IF;
                                               END_FOR;
                                               IF #m < 2 THEN
                                                   #initial := #initial + 9;
                                                   #länge := #länge + 9;
                                               END_IF;
                                           END_FOR;
                                       END_REGION
                                       //Feldchen 73
                                   72:
                                       REGION Feldchen 73
                                           //Beschränkung mögliche Nummer in der Zeile 9
                                           FOR #i := 72 TO 80 BY 1 DO
                                               IF #gitter[#k].nummer > 0 THEN
                                                   #gitter[#i].potenz_nummer[#gitter[#k].nummer - 1] := FALSE;
                                               END_IF;
                                           END_FOR;
                                           //Beschränkung mögliche Nummer in der Säule 1
                                           FOR #i := 0 TO 80 BY 9 DO
                                               IF #gitter[#k].nummer > 0 THEN
                                                   #gitter[#i].potenz_nummer[#gitter[#k].nummer - 1] := FALSE;
                                               END_IF;
                                           END_FOR;
                                           //Beschränkung mögliche Nummer in dem Viereck 7
                                           #initial := 54;
                                           #länge := 56;
                                           FOR #m := 0 TO 2 BY 1 DO
                                               FOR #i := #initial TO #länge BY 1 DO
                                                   IF #gitter[#k].nummer > 0 THEN
                                                       #gitter[#i].potenz_nummer[#gitter[#k].nummer - 1] := FALSE;
                                                   END_IF;
                                               END_FOR;
                                               IF #m < 2 THEN
                                                   #initial := #initial + 9;
                                                   #länge := #länge + 9;
                                               END_IF;
                                           END_FOR;
                                       END_REGION
                                       //Feldchen 74
                                   73:
                                       REGION Feldchen 74
                                           //Beschränkung mögliche Nummer in der Zeile 9
                                           FOR #i := 72 TO 80 BY 1 DO
                                               IF #gitter[#k].nummer > 0 THEN
                                                   #gitter[#i].potenz_nummer[#gitter[#k].nummer - 1] := FALSE;
                                               END_IF;
                                           END_FOR;
                                           //Beschränkung mögliche Nummer in der Säule 2
                                           FOR #i := 1 TO 80 BY 9 DO
                                               IF #gitter[#k].nummer > 0 THEN
                                                   #gitter[#i].potenz_nummer[#gitter[#k].nummer - 1] := FALSE;
                                               END_IF;
                                           END_FOR;
                                           //Beschränkung mögliche Nummer in dem Viereck 7
                                           #initial := 54;
                                           #länge := 56;
                                           FOR #m := 0 TO 2 BY 1 DO
                                               FOR #i := #initial TO #länge BY 1 DO
                                                   IF #gitter[#k].nummer > 0 THEN
                                                       #gitter[#i].potenz_nummer[#gitter[#k].nummer - 1] := FALSE;
                                                   END_IF;
                                               END_FOR;
                                               IF #m < 2 THEN
                                                   #initial := #initial + 9;
                                                   #länge := #länge + 9;
                                               END_IF;
                                           END_FOR;
                                       END_REGION
                                       //Feldchen 75
                                   74:
                                       REGION Feldchen 75
                                           //Beschränkung mögliche Nummer in der Zeile 9
                                           FOR #i := 72 TO 80 BY 1 DO
                                               IF #gitter[#k].nummer > 0 THEN
                                                   #gitter[#i].potenz_nummer[#gitter[#k].nummer - 1] := FALSE;
                                               END_IF;
                                           END_FOR;
                                           //Beschränkung mögliche Nummer in der Säule 3
                                           FOR #i := 2 TO 80 BY 9 DO
                                               IF #gitter[#k].nummer > 0 THEN
                                                   #gitter[#i].potenz_nummer[#gitter[#k].nummer - 1] := FALSE;
                                               END_IF;
                                           END_FOR;
                                           //Beschränkung mögliche Nummer in dem Viereck 7
                                           #initial := 54;
                                           #länge := 56;
                                           FOR #m := 0 TO 2 BY 1 DO
                                               FOR #i := #initial TO #länge BY 1 DO
                                                   IF #gitter[#k].nummer > 0 THEN
                                                       #gitter[#i].potenz_nummer[#gitter[#k].nummer - 1] := FALSE;
                                                   END_IF;
                                               END_FOR;
                                               IF #m < 2 THEN
                                                   #initial := #initial + 9;
                                                   #länge := #länge + 9;
                                               END_IF;
                                           END_FOR;
                                       END_REGION
                                       //Feldchen 76
                                   75:
                                       REGION Feldchen 76
                                           //Beschränkung mögliche Nummer in der Zeile 9
                                           FOR #i := 72 TO 80 BY 1 DO
                                               IF #gitter[#k].nummer > 0 THEN
                                                   #gitter[#i].potenz_nummer[#gitter[#k].nummer - 1] := FALSE;
                                               END_IF;
                                           END_FOR;
                                           //Beschränkung mögliche Nummer in der Säule 4
                                           FOR #i := 3 TO 80 BY 9 DO
                                               IF #gitter[#k].nummer > 0 THEN
                                                   #gitter[#i].potenz_nummer[#gitter[#k].nummer - 1] := FALSE;
                                               END_IF;
                                           END_FOR;
                                           //Beschränkung mögliche Nummer in dem Viereck 8
                                           #initial := 57;
                                           #länge := 59;
                                           FOR #m := 0 TO 2 BY 1 DO
                                               FOR #i := #initial TO #länge BY 1 DO
                                                   IF #gitter[#k].nummer > 0 THEN
                                                       #gitter[#i].potenz_nummer[#gitter[#k].nummer - 1] := FALSE;
                                                   END_IF;
                                               END_FOR;
                                               IF #m < 2 THEN
                                                   #initial := #initial + 9;
                                                   #länge := #länge + 9;
                                               END_IF;
                                           END_FOR;
                                       END_REGION
                                       //Feldchen 77
                                   76:
                                       REGION Feldchen 77
                                           //Beschränkung mögliche Nummer in der Zeile 9
                                           FOR #i := 72 TO 80 BY 1 DO
                                               IF #gitter[#k].nummer > 0 THEN
                                                   #gitter[#i].potenz_nummer[#gitter[#k].nummer - 1] := FALSE;
                                               END_IF;
                                           END_FOR;
                                           //Beschränkung mögliche Nummer in der Säule 5
                                           FOR #i := 4 TO 80 BY 9 DO
                                               IF #gitter[#k].nummer > 0 THEN
                                                   #gitter[#i].potenz_nummer[#gitter[#k].nummer - 1] := FALSE;
                                               END_IF;
                                           END_FOR;
                                           //Beschränkung mögliche Nummer in dem Viereck 8
                                           #initial := 57;
                                           #länge := 59;
                                           FOR #m := 0 TO 2 BY 1 DO
                                               FOR #i := #initial TO #länge BY 1 DO
                                                   IF #gitter[#k].nummer > 0 THEN
                                                       #gitter[#i].potenz_nummer[#gitter[#k].nummer - 1] := FALSE;
                                                   END_IF;
                                               END_FOR;
                                               IF #m < 2 THEN
                                                   #initial := #initial + 9;
                                                   #länge := #länge + 9;
                                               END_IF;
                                           END_FOR;
                                       END_REGION
                                       //Feldchen 78
                                   77:
                                       REGION Feldchen 78
                                           //Beschränkung mögliche Nummer in der Zeile 9
                                           FOR #i := 72 TO 80 BY 1 DO
                                               IF #gitter[#k].nummer > 0 THEN
                                                   #gitter[#i].potenz_nummer[#gitter[#k].nummer - 1] := FALSE;
                                               END_IF;
                                           END_FOR;
                                           //Beschränkung mögliche Nummer in der Säule 6
                                           FOR #i := 5 TO 80 BY 9 DO
                                               IF #gitter[#k].nummer > 0 THEN
                                                   #gitter[#i].potenz_nummer[#gitter[#k].nummer - 1] := FALSE;
                                               END_IF;
                                           END_FOR;
                                           //Beschränkung mögliche Nummer in dem Viereck 8
                                           #initial := 57;
                                           #länge := 59;
                                           FOR #m := 0 TO 2 BY 1 DO
                                               FOR #i := #initial TO #länge BY 1 DO
                                                   IF #gitter[#k].nummer > 0 THEN
                                                       #gitter[#i].potenz_nummer[#gitter[#k].nummer - 1] := FALSE;
                                                   END_IF;
                                               END_FOR;
                                               IF #m < 2 THEN
                                                   #initial := #initial + 9;
                                                   #länge := #länge + 9;
                                               END_IF;
                                           END_FOR;
                                       END_REGION
                                       //Feldchen 79
                                   78:
                                       REGION Feldchen 79
                                           //Beschränkung mögliche Nummer in der Zeile 9
                                           FOR #i := 72 TO 80 BY 1 DO
                                               IF #gitter[#k].nummer > 0 THEN
                                                   #gitter[#i].potenz_nummer[#gitter[#k].nummer - 1] := FALSE;
                                               END_IF;
                                           END_FOR;
                                           //Beschränkung mögliche Nummer in der Säule 7
                                           FOR #i := 6 TO 80 BY 9 DO
                                               IF #gitter[#k].nummer > 0 THEN
                                                   #gitter[#i].potenz_nummer[#gitter[#k].nummer - 1] := FALSE;
                                               END_IF;
                                           END_FOR;
                                           //Beschränkung mögliche Nummer in dem Viereck 9
                                           #initial := 60;
                                           #länge := 62;
                                           FOR #m := 0 TO 2 BY 1 DO
                                               FOR #i := #initial TO #länge BY 1 DO
                                                   IF #gitter[#k].nummer > 0 THEN
                                                       #gitter[#i].potenz_nummer[#gitter[#k].nummer - 1] := FALSE;
                                                   END_IF;
                                               END_FOR;
                                               IF #m < 2 THEN
                                                   #initial := #initial + 9;
                                                   #länge := #länge + 9;
                                               END_IF;
                                           END_FOR;
                                       END_REGION
                                       //Feldchen 80
                                   79:
                                       REGION Feldchen 80
                                           //Beschränkung mögliche Nummer in der Zeile 9
                                           FOR #i := 72 TO 80 BY 1 DO
                                               IF #gitter[#k].nummer > 0 THEN
                                                   #gitter[#i].potenz_nummer[#gitter[#k].nummer - 1] := FALSE;
                                               END_IF;
                                           END_FOR;
                                           //Beschränkung mögliche Nummer in der Säule 8
                                           FOR #i := 7 TO 80 BY 9 DO
                                               IF #gitter[#k].nummer > 0 THEN
                                                   #gitter[#i].potenz_nummer[#gitter[#k].nummer - 1] := FALSE;
                                               END_IF;
                                           END_FOR;
                                           //Beschränkung mögliche Nummer in dem Viereck 9
                                           #initial := 60;
                                           #länge := 62;
                                           FOR #m := 0 TO 2 BY 1 DO
                                               FOR #i := #initial TO #länge BY 1 DO
                                                   IF #gitter[#k].nummer > 0 THEN
                                                       #gitter[#i].potenz_nummer[#gitter[#k].nummer - 1] := FALSE;
                                                   END_IF;
                                               END_FOR;
                                               IF #m < 2 THEN
                                                   #initial := #initial + 9;
                                                   #länge := #länge + 9;
                                               END_IF;
                                           END_FOR;
                                       END_REGION
                                       //Feldchen 81
                                   80:
                                       REGION Feldchen 81
                                           //Beschränkung mögliche Nummer in der Zeile 9
                                           FOR #i := 72 TO 80 BY 1 DO
                                               IF #gitter[#k].nummer > 0 THEN
                                                   #gitter[#i].potenz_nummer[#gitter[#k].nummer - 1] := FALSE;
                                               END_IF;
                                           END_FOR;
                                           //Beschränkung mögliche Nummer in der Säule 9
                                           FOR #i := 8 TO 80 BY 9 DO
                                               IF #gitter[#k].nummer > 0 THEN
                                                   #gitter[#i].potenz_nummer[#gitter[#k].nummer - 1] := FALSE;
                                               END_IF;
                                           END_FOR;
                                           //Beschränkung mögliche Nummer in dem Viereck 9
                                           #initial := 60;
                                           #länge := 62;
                                           FOR #m := 0 TO 2 BY 1 DO
                                               FOR #i := #initial TO #länge BY 1 DO
                                                   IF #gitter[#k].nummer > 0 THEN
                                                       #gitter[#i].potenz_nummer[#gitter[#k].nummer - 1] := FALSE;
                                                   END_IF;
                                               END_FOR;
                                               IF #m < 2 THEN
                                                   #initial := #initial + 9;
                                                   #länge := #länge + 9;
                                               END_IF;
                                           END_FOR;
                                       END_REGION
                               END_CASE;
                           END_REGION
                       END_IF;
                   END_REGION
                   REGION Letze Nummer und Möglichkeiten Feld aufschreiben
                       //Letze Nummer und Möglichkeiten Feld nach jeder Schleife aufschreiben
                       FOR #i := 0 TO 80 BY 1 DO
                           #gitter_letzte_num[#i].nummer := #gitter[#i].nummer;
                           FOR #j := 0 TO 8 BY 1 DO
                               #gitter_letzte_num[#i].potenz_nummer[#j] := #gitter[#i].potenz_nummer[#j];
                           END_FOR;
                       END_FOR;
                   END_REGION
               END_FOR;
           END_IF;
       END_REGION
   END_REGION
END_FUNCTION_BLOCK

(* ===== HMI "HMI_RT_1" =====
system functions are stored by id; their names below are inferred from use

ScreenModuleEditorView "BB_Sudoku" 640x480
   Group "gitter" at 163,83 size 315x315; FormatPattern 9
   Button "aktualisierung_taster" at 133,21 size 45x45; TextOff 'Text'; PictureOff "refresh"
      on Release: InvertBit("HMI.aktualisierung_taster")
      on Press: InvertBit("HMI.aktualisierung_taster")
   Group "gitter_ohne_feld" at 163,83 size 315x315
   IOField "EA-Feld_0" at 166,85 size 30x32; FormatPattern ?
      ProcessValue <- "HMI.gitter[0]"
   IOField "EA-Feld_1" at 201,85 size 30x32; FormatPattern ?
      ProcessValue <- "HMI.gitter[1]"
   IOField "EA-Feld_2" at 236,85 size 30x32; FormatPattern ?
      ProcessValue <- "HMI.gitter[2]"
   IOField "EA-Feld_3" at 271,85 size 30x32; FormatPattern ?
      ProcessValue <- "HMI.gitter[3]"
   IOField "EA-Feld_4" at 306,85 size 30x32; FormatPattern ?
      ProcessValue <- "HMI.gitter[4]"
   IOField "EA-Feld_5" at 341,85 size 30x32; FormatPattern ?
      ProcessValue <- "HMI.gitter[5]"
   IOField "EA-Feld_6" at 376,85 size 30x32; FormatPattern ?
      ProcessValue <- "HMI.gitter[6]"
   IOField "EA-Feld_7" at 411,85 size 30x32; FormatPattern ?
      ProcessValue <- "HMI.gitter[7]"
   IOField "EA-Feld_8" at 446,85 size 30x32; FormatPattern ?
      ProcessValue <- "HMI.gitter[8]"
   IOField "EA-Feld_17" at 446,120 size 30x32; FormatPattern ?
      ProcessValue <- "HMI.gitter[17]"
   IOField "EA-Feld_26" at 446,155 size 30x32; FormatPattern ?
      ProcessValue <- "HMI.gitter[26]"
   IOField "EA-Feld_35" at 446,190 size 30x32; FormatPattern ?
      ProcessValue <- "HMI.gitter[35]"
   IOField "EA-Feld_44" at 446,225 size 30x32; FormatPattern ?
      ProcessValue <- "HMI.gitter[44]"
   IOField "EA-Feld_53" at 446,260 size 30x32; FormatPattern ?
      ProcessValue <- "HMI.gitter[53]"
   IOField "EA-Feld_62" at 446,295 size 30x32; FormatPattern ?
      ProcessValue <- "HMI.gitter[62]"
   IOField "EA-Feld_71" at 446,330 size 30x32; FormatPattern ?
      ProcessValue <- "HMI.gitter[71]"
   IOField "EA-Feld_80" at 446,365 size 30x32; FormatPattern ?
      ProcessValue <- "HMI.gitter[80]"
   IOField "EA-Feld_16" at 411,120 size 30x32; FormatPattern ?
      ProcessValue <- "HMI.gitter[16]"
   IOField "EA-Feld_25" at 411,155 size 30x32; FormatPattern ?
      ProcessValue <- "HMI.gitter[25]"
   IOField "EA-Feld_15" at 376,120 size 30x32; FormatPattern ?
      ProcessValue <- "HMI.gitter[15]"
   IOField "EA-Feld_34" at 411,190 size 30x32; FormatPattern ?
      ProcessValue <- "HMI.gitter[34]"
   IOField "EA-Feld_43" at 411,225 size 30x32; FormatPattern ?
      ProcessValue <- "HMI.gitter[43]"
   IOField "EA-Feld_52" at 411,260 size 30x32; FormatPattern ?
      ProcessValue <- "HMI.gitter[52]"
   IOField "EA-Feld_61" at 411,295 size 30x32; FormatPattern ?
      ProcessValue <- "HMI.gitter[61]"
   IOField "EA-Feld_70" at 411,330 size 30x32; FormatPattern ?
      ProcessValue <- "HMI.gitter[70]"
   IOField "EA-Feld_79" at 411,365 size 30x32; FormatPattern ?
      ProcessValue <- "HMI.gitter[79]"
   IOField "EA-Feld_69" at 376,330 size 30x32; FormatPattern ?
      ProcessValue <- "HMI.gitter[69]"
   IOField "EA-Feld_78" at 376,365 size 30x32; FormatPattern ?
      ProcessValue <- "HMI.gitter[78]"
   IOField "EA-Feld_60" at 376,295 size 30x32; FormatPattern ?
      ProcessValue <- "HMI.gitter[60]"
   IOField "EA-Feld_33" at 376,190 size 30x32; FormatPattern ?
      ProcessValue <- "HMI.gitter[33]"
   IOField "EA-Feld_24" at 376,155 size 30x32; FormatPattern ?
      ProcessValue <- "HMI.gitter[24]"
   IOField "EA-Feld_41" at 341,225 size 30x32; FormatPattern ?
      ProcessValue <- "HMI.gitter[41]"
   IOField "EA-Feld_32" at 341,190 size 30x32; FormatPattern ?
      ProcessValue <- "HMI.gitter[32]"
   IOField "EA-Feld_42" at 376,225 size 30x32; FormatPattern ?
      ProcessValue <- "HMI.gitter[42]"
   IOField "EA-Feld_13" at 306,120 size 30x32; FormatPattern ?
      ProcessValue <- "HMI.gitter[13]"
   IOField "EA-Feld_31" at 306,190 size 30x32; FormatPattern ?
      ProcessValue <- "HMI.gitter[31]"
   IOField "EA-Feld_56" at 236,295 size 30x32; FormatPattern ?
      ProcessValue <- "HMI.gitter[56]"
   IOField "EA-Feld_54" at 166,295 size 30x32; FormatPattern ?
      ProcessValue <- "HMI.gitter[54]"
   IOField "EA-Feld_27" at 166,190 size 30x32; FormatPattern ?
      ProcessValue <- "HMI.gitter[27]"
   IOField "EA-Feld_45" at 166,260 size 30x32; FormatPattern ?
      ProcessValue <- "HMI.gitter[45]"
   IOField "EA-Feld_18" at 166,155 size 30x32; FormatPattern ?
      ProcessValue <- "HMI.gitter[18]"
   IOField "EA-Feld_9" at 166,120 size 30x32; FormatPattern ?
      ProcessValue <- "HMI.gitter[9]"
   IOField "EA-Feld_63" at 166,330 size 30x32; FormatPattern ?
      ProcessValue <- "HMI.gitter[63]"
   IOField "EA-Feld_72" at 166,365 size 30x32; FormatPattern ?
      ProcessValue <- "HMI.gitter[72]"
   IOField "EA-Feld_36" at 166,225 size 30x32; FormatPattern ?
      ProcessValue <- "HMI.gitter[36]"
   IOField "EA-Feld_30" at 271,190 size 30x32; FormatPattern ?
      ProcessValue <- "HMI.gitter[30]"
   IOField "EA-Feld_12" at 271,120 size 30x32; FormatPattern ?
      ProcessValue <- "HMI.gitter[12]"
   IOField "EA-Feld_67" at 306,330 size 30x32; FormatPattern ?
      ProcessValue <- "HMI.gitter[67]"
   IOField "EA-Feld_50" at 341,260 size 30x32; FormatPattern ?
      ProcessValue <- "HMI.gitter[50]"
   IOField "EA-Feld_51" at 376,260 size 30x32; FormatPattern ?
      ProcessValue <- "HMI.gitter[51]"
   IOField "EA-Feld_37" at 201,225 size 30x32; FormatPattern ?
      ProcessValue <- "HMI.gitter[37]"
   IOField "EA-Feld_38" at 236,225 size 30x32; FormatPattern ?
      ProcessValue <- "HMI.gitter[38]"
   IOField "EA-Feld_39" at 271,225 size 30x32; FormatPattern ?
      ProcessValue <- "HMI.gitter[39]"
   IOField "EA-Feld_58" at 306,295 size 30x32; FormatPattern ?
      ProcessValue <- "HMI.gitter[58]"
   IOField "EA-Feld_40" at 306,225 size 30x32; FormatPattern ?
      ProcessValue <- "HMI.gitter[40]"
   IOField "EA-Feld_49" at 306,260 size 30x32; FormatPattern ?
      ProcessValue <- "HMI.gitter[49]"
   IOField "EA-Feld_48" at 271,260 size 30x32; FormatPattern ?
      ProcessValue <- "HMI.gitter[48]"
   IOField "EA-Feld_59" at 341,295 size 30x32; FormatPattern ?
      ProcessValue <- "HMI.gitter[59]"
   IOField "EA-Feld_65" at 236,330 size 30x32; FormatPattern ?
      ProcessValue <- "HMI.gitter[65]"
   IOField "EA-Feld_28" at 201,190 size 30x32; FormatPattern ?
      ProcessValue <- "HMI.gitter[28]"
   IOField "EA-Feld_76" at 306,365 size 30x32; FormatPattern ?
      ProcessValue <- "HMI.gitter[76]"
   IOField "EA-Feld_66" at 271,330 size 30x32; FormatPattern ?
      ProcessValue <- "HMI.gitter[66]"
   IOField "EA-Feld_57" at 271,295 size 30x32; FormatPattern ?
      ProcessValue <- "HMI.gitter[57]"
   IOField "EA-Feld_68" at 341,330 size 30x32; FormatPattern ?
      ProcessValue <- "HMI.gitter[68]"
   IOField "EA-Feld_77" at 341,365 size 30x32; FormatPattern ?
      ProcessValue <- "HMI.gitter[77]"
   IOField "EA-Feld_75" at 271,365 size 30x32; FormatPattern ?
      ProcessValue <- "HMI.gitter[75]"
   IOField "EA-Feld_74" at 236,365 size 30x32; FormatPattern ?
      ProcessValue <- "HMI.gitter[74]"
   IOField "EA-Feld_14" at 341,120 size 30x32; FormatPattern ?
      ProcessValue <- "HMI.gitter[14]"
   IOField "EA-Feld_22" at 306,155 size 30x32; FormatPattern ?
      ProcessValue <- "HMI.gitter[22]"
   IOField "EA-Feld_21" at 271,155 size 30x32; FormatPattern ?
      ProcessValue <- "HMI.gitter[21]"
   IOField "EA-Feld_23" at 341,155 size 30x32; FormatPattern ?
      ProcessValue <- "HMI.gitter[23]"
   IOField "EA-Feld_29" at 236,190 size 30x32; FormatPattern ?
      ProcessValue <- "HMI.gitter[29]"
   IOField "EA-Feld_20" at 236,155 size 30x32; FormatPattern ?
      ProcessValue <- "HMI.gitter[20]"
   IOField "EA-Feld_11" at 236,120 size 30x32; FormatPattern ?
      ProcessValue <- "HMI.gitter[11]"
   IOField "EA-Feld_10" at 201,120 size 30x32; FormatPattern ?
      ProcessValue <- "HMI.gitter[10]"
   IOField "EA-Feld_19" at 201,155 size 30x32; FormatPattern ?
      ProcessValue <- "HMI.gitter[19]"
   IOField "EA-Feld_46" at 201,260 size 30x32; FormatPattern ?
      ProcessValue <- "HMI.gitter[46]"
   IOField "EA-Feld_47" at 236,260 size 30x32; FormatPattern ?
      ProcessValue <- "HMI.gitter[47]"
   IOField "EA-Feld_55" at 201,295 size 30x32; FormatPattern ?
      ProcessValue <- "HMI.gitter[55]"
   IOField "EA-Feld_64" at 201,330 size 30x32; FormatPattern ?
      ProcessValue <- "HMI.gitter[64]"
   IOField "EA-Feld_73" at 201,365 size 30x32; FormatPattern ?
      ProcessValue <- "HMI.gitter[73]"
   Group "Linien" at 163,83 size 315x315
*)